{attribute 'no_explicit_call'} 
FUNCTION_BLOCK PUBLIC FB_ListSTRING IMPLEMENTS I_ListSTRING
VAR
	pList: 			POINTER TO STRING(255);
	nLength:		DINT;
	aList:			POINTER TO POINTER TO ARRAY [0..100] OF STRING(255):=ADR(pList);
END_VAR

METHOD FB_exit : BOOL
VAR_INPUT
	bInCopyCode : BOOL; // if TRUE, the exit method is called for exiting an instance that is copied afterwards (online change).
END_VAR
M_Clear();
END_METHOD

METHOD M_Add : BOOL
VAR_INPUT
	Value:		STRING(255);
END_VAR
VAR
	pOldList: 	POINTER TO STRING(255);
END_VAR
// First Item
IF pList = 0 THEN
	nLength:= nLength + 1;
	pList:= __NEW(POINTER TO STRING(255), SIZEOF(STRING(255)));
ELSE
	// backup 
	pOldList:= pList;
	// new Length
	nLength:= nLength + 1;
	// new pointer
	pList:= __NEW(POINTER TO STRING(255),DINT_TO_UDINT(SIZEOF(STRING(255)) * nLength));
	// restore
	Memcpy(pList,pOldList, DINT_TO_UDINT(SIZEOF(STRING(255)) *(nLength -1)));
	// delete old
	__DELETE(pOldList);
END_IF

// add new Object
pList[nLength-1]:= Value;
M_Add:= TRUE;
END_METHOD

METHOD M_Clear : BOOL
IF pList <> 0 THEN
	nLength:= 0;
	__DELETE(pList);
	M_Clear:= TRUE;
END_IF
END_METHOD

METHOD M_Index : DINT
VAR_INPUT
	Value:	STRING(255);
END_VAR
VAR
	nIndex: 	DINT;
END_VAR
// Object already in List
M_Index := -1;
WHILE nIndex < nLength DO
  IF pList[nIndex] = Value THEN
        M_Index := nIndex;
        RETURN;
    END_IF
	nIndex := nIndex + 1;
END_WHILE
END_METHOD

METHOD PUBLIC M_Insert : BOOL
VAR_INPUT
	Position:		UDINT;
	Value:			STRING(255);
END_VAR
VAR
	pOldList: 		POINTER TO STRING(255);
END_VAR
IF nLength > Position THEN
	// backup 
	pOldList:= pList;
	// new Length
	nLength:= nLength + 1;
	// new pointer
	pList:= __NEW(POINTER TO STRING(255),DINT_TO_UDINT(SIZEOF(STRING(255)) * nLength));
	// restore
	Memcpy(pList, pOldList, DINT_TO_UDINT(SIZEOF(STRING(255)) *(nLength -1)));
	MemMove(pList + DINT_TO_UDINT(SIZEOF(STRING(255)) * (Position + 1)), pList + DINT_TO_UDINT(SIZEOF(STRING(255)) * Position), DINT_TO_UDINT(SIZEOF(STRING(255)) * (nLength - Position + 1)));
	// delete old
	__DELETE(pOldList);
ELSE
	M_Insert:= FALSE;	
	RETURN;
END_IF
// add new Object
pList[Position]:= Value;
M_Insert:= TRUE;
END_METHOD

METHOD M_Item : STRING(255)
VAR_INPUT
	Index: 	DINT;
END_VAR
IF Index < (nLength) THEN
	M_Item:= pList[Index];
END_IF
END_METHOD

METHOD M_Remove : BOOL
VAR_INPUT
	Position:			DINT;
END_VAR
VAR
	pOldList:			POINTER TO STRING(255);
END_VAR
// First Item
IF nLength >= Position THEN
	// backup 
	pOldList:= pList;
	// new Length
	nLength:= nLength -1;
	// new pointer
	pList:= __NEW(POINTER TO STRING(255),DINT_TO_UDINT(SIZEOF(STRING(255)) * nLength));
	// restore lower part
	Memcpy(pList,pOldList, SIZEOF(POINTER TO STRING(255)) * DINT_TO_UDINT(Position));
	//pList[nPosition]:= iObject;
	Memcpy(pList + (SIZEOF(STRING(255))*Position),pOldList + (SIZEOF(STRING(255))*(Position + 1)), SIZEOF(STRING(255)) * DINT_TO_UDINT(nLength - Position));
	// delete old
	__DELETE(pOldList);
ELSE
	M_Remove:= FALSE;	
	RETURN;
END_IF
M_Remove:= TRUE;
END_METHOD

METHOD M_Search : DINT
VAR_INPUT
	Value:		STRING(255);
END_VAR
VAR
	nIndex: 	UINT;
END_VAR
// Object already in List
M_Search := -1;
WHILE nIndex < nLength DO
    IF pList[nIndex] = Value THEN
        M_Search := nIndex;
        RETURN;
    END_IF
	nIndex := nIndex + 1;
END_WHILE
END_METHOD

PROPERTY P_Length : DINT
GET
P_Length:= nLength;
END_GET
END_PROPERTY

END_FUNCTION_BLOCK

(* stored: Version 1.1.0.1
   POU FB_ListSTRING: Id {a989d5e2-1cf5-0358-2412-01f34683c5c9}, SpecialFunc None
   Method FB_exit: Id {9a1b1e03-9c79-04ae-0e47-529adbf0eb35}
   Method M_Add: Id {fc95c475-02ce-0a23-3d94-22fd0ca885a7}
   Method M_Clear: Id {0696c9f2-3368-02c7-3570-914b538477bb}
   Method M_Index: Id {f499fc6d-d45b-0ca4-2495-d9d9df4f4408}
   Method M_Insert: Id {6d66fd7b-af1e-0a73-0590-29550cb06d1b}
   Method M_Item: Id {29e4159c-eed0-0b05-05f7-6ee207ca7daf}
   Method M_Remove: Id {e45f8add-9693-0801-3102-f3924d7fbe37}
   Method M_Search: Id {9af81950-5ba8-0340-3e5f-5b6e67170a1c}
   Property P_Length: Id {4be58bcd-8d3b-06e7-25c0-02f6b9f73cce}
   Get Get: Id {ebd53a4d-532d-0f16-0572-d7a706cbf043} *)
